PROGRAM MAIN
VAR
	//stThisIsOurFirstInstanceOfAStructure: ST_Event;
	bBoolean: BOOL:= FALSE;
	//n: INT;
	//trigger: BOOL;
	
	
	//LocalSystemTime: FB_LocalSystemTime();
		//timeStruct: TIMESTRUCT;
	CSVPersistentEventStorage: FB_CSVPersistentEventStorage;	
	Eventlogger:Eventlogger(CSVPersistentEventStorage);
	
	//SQLPersistentEventStorage: SQLPersistentEventStorage;
	//Eventlogger2:Eventlogger(SQLPersistentEventStorage);
	
	eEventType: E_EventType:=E_EventType.Alarm ;
	eEventSeverity: TcEventSeverity:=TcEventSeverity.Critical;
	nEventIdentity: UDINT:=1;
	sEventText: STRING(255):= 'Allvarligt fel';

END_VAR

IF NOT bBoolean THEN
	Eventlogger.AddEvent(eEventType:= eEventType,eEventSeverity:= eEventSeverity,nEventIdentity:=nEventIdentity,sEventText:=sEventText);
	
	bBoolean:= TRUE;
END_IF


CSVPersistentEventStorage();

//LocalSystemTime(bEnable:=TRUE,systemTime=> timeStruct);

//stThisIsOurFirstInstanceOfAStructure.dtTimeStamp := SYSTEMTIME_TO_DT(TIMESTR:=timeStruct);
//stThisIsOurFirstInstanceOfAStructure.sEventText:= 'TEST';

END_PROGRAM

(* stored: Version 1.1.0.1, ProductVersion 3.1.4024.11
   POU MAIN: Id {336a9b16-1fa5-4eed-90ef-5a17914deabf}, SpecialFunc None *)
